// TIA Portal V18 export
TYPE "MEStoPLC_ST350"
// stored: IsFailsafeCompliant false
   STRUCT
      Common { S7_SetPoint := 'True'} : "MEStoPLC_Common";   // MES反馈公共区
      MainCheckIn { S7_SetPoint := 'True'} : "MEStoPLC_MainCheckIn";   // MES反馈主件查询结果
      SubCheckIn { S7_SetPoint := 'True'} : "MEStoPLC_SubCheckIn";   // MES反馈子件查询结果
      Processing { S7_SetPoint := 'True'} : "MEStoPLC_ProcessingExchange";   // MES反馈Processing记录结果
      MainCheckOut { S7_SetPoint := 'True'} : "MEStoPLC_MainCheckOut";   // MES反馈主件保存结果
      PrintExchange { S7_SetPoint := 'True'} : "MEStoPLC_PrintExchange";   // MES反馈打印数据
      AGVExchange { S7_SetPoint := 'True'} : "MEStoPLC_AGVExchange";   // MES反馈AGV查询结果
      RecipeData { S7_SetPoint := 'True'} : "MEStoPLC_RecipeData_OP220";   // MES反馈配方参数数据
   END_STRUCT;
END_TYPE
